// TIA Portal project "LeitungszuordnungsTester" (V14)

(* hardware
DEVICE "S7-1200-Station_1"  S7-1200 Station
   slot 0: "Baugruppenträger_0"  Rack  V1.0
   slot 1: "PLC"  CPU 1214C DC/DC/DC  6ES7 214-1AG40-0XB0  V4.1
   slot 3: "AQ 1x12BIT_1"  6ES7 232-4HA30-0XB0  V1.0
DEVICE "HMI"  KTP700 Basic PN
   slot 0: "HMI"  HMI  6AV2 123-2GB03-0AX0  13.0.1.0
   slot 1: "HMI_RT_1"  KTP700 Basic PN  6AV2 123-2GB03-0AX0  13.0.1.0
   slot 5: "HMI.IE_CP_1"  PROFINET Schnittstelle
      slot 1: "PROFINET Schnittstelle_1"  PROFINET Schnittstelle
         slot 1: "Port_1"  Port
*)

// ===== PLC "PLC"  CPU 1214C DC/DC/DC =====

VAR_GLOBAL   // PLC tag table "Standard-Variablentabelle"
   "System_Byte" AT %MB100 : Byte;
   "FirstScan" AT %M100.0 : Bool;
   "DiagStatusUpdate" AT %M100.1 : Bool;
   "AlwaysTRUE" AT %M100.2 : Bool;
   "AlwaysFALSE" AT %M100.3 : Bool;
   "Clock_Byte" AT %MB110 : Byte;
   "Clock_10Hz" AT %M110.0 : Bool;
   "Clock_5Hz" AT %M110.1 : Bool;
   "Clock_2.5Hz" AT %M110.2 : Bool;
   "Clock_2Hz" AT %M110.3 : Bool;
   "Clock_1.25Hz" AT %M110.4 : Bool;
   "Clock_1Hz" AT %M110.5 : Bool;
   "Clock_0.625Hz" AT %M110.6 : Bool;
   "Clock_0.5Hz" AT %M110.7 : Bool;
   "x_NichtVerbunden" AT %M0.0 : Bool;
   "x_AderErkennen" AT %M0.1 : Bool;
   "x_Ader_1" AT %M0.2 : Bool;
   "x_Ader_2" AT %M0.3 : Bool;
   "x_Ader_3" AT %M0.4 : Bool;
   "x_Ader_4" AT %M0.5 : Bool;
   "x_Ader_5" AT %M0.6 : Bool;
   "x_Ader_6" AT %M0.7 : Bool;
   "x_Ader_7" AT %M1.0 : Bool;
   "x_Ader_8" AT %M1.1 : Bool;
   "TestEingang" AT %I0.0 : Bool;
   "Ader_1" AT %Q0.0 : Bool;
   "Ader_2" AT %Q0.1 : Bool;
   "Ader_3" AT %Q0.2 : Bool;
   "Ader_4" AT %Q0.3 : Bool;
   "Ader_5" AT %Q0.4 : Bool;
   "Ader_6" AT %Q0.5 : Bool;
   "Ader_7" AT %Q0.6 : Bool;
   "Ader_8" AT %Q0.7 : Bool;
   "AlleAusgänge" AT %QW0 : Word;
END_VAR

FUNCTION "fcLeitungsZuordnungsTester" : Void   // FC1, FBD
{ S7_Optimized_Access := 'TRUE' }
VERSION : 0.1
BEGIN

REGION Network 1
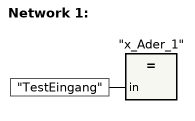
   "x_Ader_1" := "TestEingang";
END_REGION
END_FUNCTION

ORGANIZATION_BLOCK "Main"   // OB1, LAD, ProgramCycle
TITLE = "Main Program Sweep (Cycle)"
{ S7_Optimized_Access := 'TRUE' }
VERSION : 0.1
   VAR_INPUT
      Initial_Call : Bool;   // Initial call of this OB
      Remanence : Bool;   // =True, if remanent data are available
   END_VAR
BEGIN

REGION Network 1: -Q1
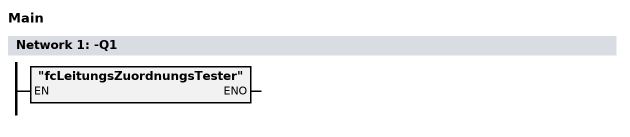
   RUNG wire#powerrail
      "fcLeitungsZuordnungsTester"()
   END_RUNG
   // the same network as SCL:
   "fcLeitungsZuordnungsTester"();
END_REGION
END_ORGANIZATION_BLOCK

ORGANIZATION_BLOCK "Startup"   // OB100, SCL, Startup
TITLE = "Complete Restart"
{ S7_Optimized_Access := 'TRUE' }
VERSION : 0.1
   VAR_INPUT
      LostRetentive : Bool;   // True if retentive data are lost
      LostRTC : Bool;   // True if date and time are lost
   END_VAR
BEGIN
   "AlleAusgänge" := 16#0000;
END_ORGANIZATION_BLOCK

(* ===== HMI "HMI_RT_1" =====
connection "HMI_Verbindung_1": ETHERNET, SMART_S7_1200_OMS

HMI tags "Standard-Variablentabelle"
   "x_NichtVerbunden" : Bool = PLC x_NichtVerbunden AT %M0.0, 100 ms
   "x_AderErkennen" : Bool = PLC x_AderErkennen AT %M0.1, 100 ms
   "x_Ader_1" : Bool = PLC x_Ader_1 AT %M0.2, 100 ms
   "x_Ader_2" : Bool = PLC x_Ader_2 AT %M0.3, 100 ms
   "x_Ader_3" : Bool = PLC x_Ader_3 AT %M0.4, 100 ms
   "x_Ader_4" : Bool = PLC x_Ader_4 AT %M0.5, 100 ms
   "x_Ader_5" : Bool = PLC x_Ader_5 AT %M0.6, 100 ms
   "x_Ader_6" : Bool = PLC x_Ader_6 AT %M0.7, 100 ms
   "x_Ader_7" : Bool = PLC x_Ader_7 AT %M1.0, 100 ms
   "x_Ader_8" : Bool = PLC x_Ader_8 AT %M1.1, 100 ms

screen "LeitungszuordnungsTester" 800x480
   TextField "Textfeld_2" at 90,0 size 641x62; Text 'Leitungszuordnungstester'
   TextField "Textfeld_3" at 187,65 size 410x23; Text 'Zu testende Leitung mit Eingang DI 0.0 verbinden'
   TextField "Textfeld_1" at 100,200 size 538x81; Text 'Nicht verbunden'
      Visibility <- "x_NichtVerbunden"
   TextField "Textfeld_4" at 100,200 size 557x81; Text 'Ader erkennen ...'
      Visibility <- "x_AderErkennen"
   TextField "Textfeld_5" at 100,200 size 510x81; Text 'Ader 4 (DQ 0.3)'
      Visibility <- "x_Ader_4"
   TextField "Textfeld_6" at 100,200 size 510x81; Text 'Ader 2 (DQ 0.1)'
      Visibility <- "x_Ader_2"
   TextField "Textfeld_7" at 100,200 size 510x81; Text 'Ader 3 (DQ 0.2)'
      Visibility <- "x_Ader_3"
   TextField "Textfeld_8" at 100,200 size 510x81; Text 'Ader 1 (DQ 0.0)'
      Visibility <- "x_Ader_1"
   TextField "Textfeld_9" at 100,200 size 510x81; Text 'Ader 6 (DQ 0.5)'
      Visibility <- "x_Ader_6"
   TextField "Textfeld_10" at 100,200 size 510x81; Text 'Ader 5 (DQ 0.4)'
      Visibility <- "x_Ader_5"
   TextField "Textfeld_11" at 100,200 size 510x81; Text 'Ader 8 (DQ 0.7)'
      Visibility <- "x_Ader_8"
   TextField "Textfeld_12" at 100,200 size 510x81; Text 'Ader 7 (DQ 0.6)'
      Visibility <- "x_Ader_7"
*)